PROGRAM POU_TestGitHub
VAR
	input : BOOL;
	output : BOOL;
END_VAR

output := input;

END_PROGRAM

(* stored: Version 1.1.0.1, ProductVersion 3.1.4024.11
   POU POU_TestGitHub: Id {b3b56a95-9553-4b01-b7d0-5e99422eb172}, SpecialFunc None *)
